// TIA Portal V20 export
TYPE "IO_DI"
   STRUCT
      IN : Struct
         Input : Bool;
      END_STRUCT;
   END_STRUCT;
END_TYPE
